// TwinCAT 3 PLC project LogicTask
// ProgramVersion: 3.1.4023.0
// libraries:
//   Tc2_Standard, * (Beckhoff Automation GmbH)
//   Tc2_System, * (Beckhoff Automation GmbH)
//   Tc3_Module, * (Beckhoff Automation GmbH)
// project tree:
//   / Fast_Task.TcTTO, PlcTask.TcTTO
//   GVLs/ GVL_Robot_IO_Map.TcGVL
//   POUs/ MAIN.TcPOU
//   RobotMapping/ RobotMapping.TcPOU
//   SafetyLogic/ EmgFunctions.TcPOU, Pulser.TcPOU
// real-time tasks:
//   TASK Fast Task: cycle T#1ms, priority 1, ADS port 351
//   TASK PlcTask: cycle T#10ms, priority 5, ADS port 352
// I/O:
//   DEVICE Device 1 (EtherCAT), AmsNetId 5.58.206.91.2.1
//     Term 1 (EK1200) [EK1200-5000 EtherCAT Power supply (2A E-Bus)]
//       Term 2 (EL1008) [EL1008 8Ch. Dig. Input 24V, 3ms]
//       Term 3 (EL2008) [EL2008 8Ch. Dig. Output 24V, 0.5A]
//       Term 4 (EL1918) [EL1918, 8Ch. Safety Input 24V, TwinSAFE]
//         modules: Module 1 (FSOE), Module 2 (FSLOGIC)
//       Term 5 (EL1918) [EL1918, 8Ch. Safety Input 24V, TwinSAFE]
//         modules: Module 1 (FSOE), Module 2 (FSLOGIC)
//       Term 6 (EL2904) [EL2904, 4 Ch. Safety Output 24V, 0.5A, TwinSAFE]
//         modules: Module 1 (FSOES), Module 2 (DO)
//       Term 7 (EL2904) [EL2904, 4 Ch. Safety Output 24V, 0.5A, TwinSAFE]
//         modules: Module 1 (FSOES), Module 2 (DO)
//       Term 8 (EK1122) BusJunction [EK1122 2 port EtherCAT junction]
//         Term 9 (EK1914) BusCoupler Boom [EK1914, 2 Ch. Safety Input/Output 24V,  TwinSAFE]
//           modules: Module 1 (FSOE), Module 2 (DIO)
//           Term 10 (EL1008) [EL1008 8Ch. Dig. Input 24V, 3ms]
//           Term 11 (EL1918) [EL1918, 8Ch. Safety Input 24V, TwinSAFE]
//             modules: Module 1 (FSOE), Module 2 (FSLOGIC)
//           Term 12 (EL1008) [EL1008 8Ch. Dig. Input 24V, 3ms]
//           Term 13 (EL9410) [EL9410 E-Bus Power Supplier  (Diagnostics)]
//           Term 14 (EL1008) [EL1008 8Ch. Dig. Input 24V, 3ms]
//           Term 15 (EL2008) [EL2008 8Ch. Dig. Output 24V, 0.5A]
//           Term 16 (EL2008) [EL2008 8Ch. Dig. Output 24V, 0.5A]
//           Term 17 (EL6751) [EL6751 CANopen Master]
//           Term 22 (EL9011) [EL9011 End Terminal]
//         Term 18 (EK1914) BusCoupler Robot [EK1914, 2 Ch. Safety Input/Output 24V,  TwinSAFE]
//           modules: Module 1 (FSOE), Module 2 (DIO)
//           Term 19 (EL3024) [EL3024 4Ch. Ana. Input 4-20mA DIFF]
//           Term 23 (EL9011) [EL9011 End Terminal]
//         Term 20 (EK1100) [EK1100 EtherCAT Coupler (2A E-Bus)]
//       Term 21 (EL6652-0010) Robot InOut [EL6652-0010 EtherNet/IP Adapter (Slave)]
//       Term 24 (EL9011) [EL9011 End Terminal]
//   DEVICE Device 3 (NOV-DP-RAM)
//   DEVICE Device 2 (EL6751) Canbus, AmsNetId 5.58.206.91.3.1
//   DEVICE Device 4 (ECAT EIP Adapter (EL6652-0010)), AmsNetId 5.58.206.91.5.1
//     Box 25 (TC EtherNet/IP Slave)
// variable links:
//   LogicTask/LogicTask Instance <-> Device 1 (EtherCAT)/Term 1 (EK1200)/Term 2 (EL1008)
//     Fast_Task Inputs/GVL_Robot_IO_Map.bInT2_PLC <-> Channel 1/Input
//     Fast_Task Inputs/GVL_Robot_IO_Map.bInT2_PLC @bit {1..7} <-> Channel {2..8}/Input  (7 links)
//   LogicTask/LogicTask Instance <-> Device 1 (EtherCAT)/Term 1 (EK1200)/Term 3 (EL2008)
//     Fast_Task Outputs/GVL_Robot_IO_Map.bOutT3_PLC <-> Channel 1/Output
//     Fast_Task Outputs/GVL_Robot_IO_Map.bOutT3_PLC @bit {1..7} <-> Channel {2..8}/Output  (7 links)
//   LogicTask/LogicTask Instance <-> Device 4 (ECAT EIP Adapter (EL6652-0010))/Box 25 (TC EtherNet/IP Slave)
//     Fast_Task Inputs/GVL_Robot_IO_Map.bInT3_EIP <-> Assembly 1 (Input/Output)/Inputs (Outputs from Robot)/ToOutputT2
//     Fast_Task Inputs/GVL_Robot_IO_Map.uintD4_B17_EIB_constate <-> Assembly 1 (Input/Output)/Inputs (Outputs from Robot)/ConnState
//     Fast_Task Outputs/GVL_Robot_IO_Map.bOutT2_EIP <-> Assembly 1 (Input/Output)/Outputs (Inputs to Robot)/FromInputT2

CONFIGURATION LogicTask
    RESOURCE PLC ON TwinCAT3
        TASK Fast_Task(INTERVAL := T#1ms, PRIORITY := 1);
        TASK PlcTask(INTERVAL := T#10ms, PRIORITY := 5);
        PROGRAM RobotMapping WITH Fast_Task : RobotMapping;
        PROGRAM MAIN WITH PlcTask : MAIN;
    END_RESOURCE
END_CONFIGURATION

// ---- GVLs/GVL_Robot_IO_Map.TcGVL
{attribute 'qualified_only'}
VAR_GLOBAL
//--- POwer Cabinet -----------
	//EL1008 (T2) Input
	bInT2_PLC 			AT %I* :BYTE;
	bOutT2_EIP 			AT %Q* :BYTE;
	
	//EL2008 (T3) Output	
	bInT3_EIP 			AT %I* :BYTE;
	bOutT3_PLC 			AT %Q* :BYTE;
	
	
//--- Status EIP -------------------
	//EL6652-0010 (T23)
	
	//EL6652 (D4-Box28) 	
	uintD4_B17_EIB_state AT %I* :UINT;
	uintD4_B17_EIB_constate AT %I* :UINT;
	
END_VAR

// ---- RobotMapping/RobotMapping.TcPOU
PROGRAM RobotMapping
VAR
	TmpByte : BYTE;
	DelayRobOffOutput : TON := (PT:=T#5S);
	TOutCom : TOF := (PT:=T#1S);
	RobotOff : BOOL := FALSE;
END_VAR

//--- If EIP communication is running -----------------
TOutCom(IN :=(GVL_Robot_Io_Map.uintD4_B17_EIB_constate = 0));

//update outputs
IF (TOutCom.Q) THEN
//--- Power Cabinet Outputs from Robot--------------------------------
	//EL2008 (T3)
	GVL_Robot_Io_Map.bOutT3_PLC 		:= GVL_Robot_Io_Map.bInT3_EIP;
	
	DelayRobOffOutput(IN := FALSE);
ELSE //--- Else write 0 to outputs
	GVL_Robot_Io_Map.bOutT3_PLC 		:= 0;
	DelayRobOffOutput(IN := TRUE);
END_IF

//--- Power Cabinet Inputs to Robot --------------------------------
	//EL1008 (T2)
GVL_Robot_Io_Map.bOutT2_EIP 		:= GVL_Robot_Io_Map.bInT2_PLC ;

END_PROGRAM

// ---- POUs/MAIN.TcPOU
PROGRAM MAIN
VAR
END_VAR

EmgFunctions();

END_PROGRAM

// ---- SafetyLogic/EmgFunctions.TcPOU
PROGRAM EmgFunctions
VAR_INPUT
	ActivateEStop2 : BOOL;	
END_VAR
VAR
	qResetEmergencyStop  AT %Q* : BOOL;
	qErrorAcknowledgement AT %Q* : BOOL;
	
	qEstopLamp AT %Q* : BOOL;
	iResetEmergencyStop  AT %I* : BOOL;
	iEstopOkFromSafety AT %I* : BOOL;
	qSafetyRun AT %Q* : BOOL;
	
	noOfBlinks : INT := 1;
	blinker : Pulser := (ShortPulseWidth:=T#200MS, LongPulseWidth:=T#3S, DeadPulseWidth:=T#150MS);
	RedBlink : Pulser := (ShortPulseWidth:=T#200MS, LongPulseWidth:=T#300MS, DeadPulseWidth:=T#200MS);
	RedBlinkFlag : BOOL;
	TmpBlink1 : BOOL;
	Pulstimer : TP;
END_VAR

qSafetyRun := TRUE;
// Reset Error in safety PLC
IF iResetEmergencyStop THEN
	Pulstimer(IN:=TRUE,PT:=T#300MS);
	qErrorAcknowledgement := PulsTimer.Q;
	TmpBlink1 := PulsTimer.Q;
//	qResetDoor1ToSafety := iZone1IsActiv; 
//	qResetDoor2ToSafety := iZone2IsActiv; 
	qResetEmergencyStop := RedBlinkFlag;
ELSE
	TmpBlink1 := FALSE;
	PulsTimer(IN:=FALSE);
	qResetEmergencyStop := FALSE;	
END_IF

END_PROGRAM

// ---- SafetyLogic/Pulser.TcPOU
FUNCTION_BLOCK Pulser
VAR_INPUT
	// Width of the counted ON pulse
	ShortPulseWidth : TIME := T#200MS;
	// Width of the paused ON pulse
	LongPulseWidth : TIME := T#2S;
	// Width of the deadtime between pulses
	DeadPulseWidth : TIME := T#300MS;
END_VAR
VAR_OUTPUT
END_VAR
VAR
END_VAR

METHOD M_Pulse : BOOL
VAR_INPUT
	// If the pulsing should be ON or OFF if OFF the return value will also be LOW/OFF
	Active : BOOL;
	// Number of short pulses
	Pulses : INT := 0;
END_VAR
VAR_INST
	pulseCounter : INT := 0;
	state : INT := 0;
	timer : TP;
END_VAR

// Return immediatly if not active.
IF NOT Active THEN
	pulseCounter := 0;
	M_Pulse := FALSE;
	state := 0;
	timer(IN:=FALSE);
	RETURN;
END_IF

// special case if 0 pulses are requested
IF Pulses <= 0 THEN
	pulseCounter := 0;
	M_Pulse := TRUE;
	state := 0;
	timer(IN:=FALSE);
	RETURN;
END_IF


CASE state OF
0: // Start the timer for high signal
	M_Pulse := TRUE;
	timer(IN:=TRUE,PT:=LongPulseWidth);
	state := 1;
1: // alive time
	IF timer.Q THEN // Keep high
		M_Pulse := TRUE;
		timer(IN:=FALSE);
	ELSE // start timer for low periode
		M_Pulse := FALSE;
		timer(IN:=TRUE,PT:=DeadPulseWidth);
		state := 2;		
	END_IF
2: // deadtime
	IF timer.Q THEN // keep low
		M_Pulse := FALSE;
		timer(IN:=FALSE);
	ELSE // start timer for high periode
		M_Pulse := TRUE;
		pulseCounter := pulseCounter + 1;
		IF pulseCounter >= Pulses THEN
			pulseCounter := 0;
			timer(IN:=TRUE,PT:=LongPulseWidth);
		ELSE
			timer(IN:=TRUE,PT:=ShortPulseWidth);
		END_IF
		state := 1;		
	END_IF
END_CASE
END_METHOD

END_FUNCTION_BLOCK
